// NETWORK 20
// label: (*IN1601 节能蓄能器气压*)
SaveEngine_PAtomsPre(
    INPUT := GVL_SaveEngine.AI_PAtomsPreMv,
    NEGFULL := PAR_HydOilPress_NegFull,
    POSFULL := PAR_HydOilPress_PosFull,
    RANGE := 400,
    Sensor_Error_LOW => CANO_SensorError_PAtomsPre,
    Sensor_Error_HIGH => CANO_SensorError_PAtomsPre); // PRESSURE
GVL_SaveEngine.AI_PAtomsPre := SaveEngine_PAtomsPre.OUTPUT;

// NETWORK 21
// IN 1602 主卷马达下降出口压力M1
SaveEngine_PM1Pre(
    INPUT := GVL_SaveEngine.AI_PM1PreMv,
    NEGFULL := PAR_HydOilPress_NegFull,
    POSFULL := PAR_HydOilPress_PosFull,
    RANGE := 400,
    Sensor_Error_LOW => CANO_SensorError_PM1,
    Sensor_Error_HIGH => CANO_SensorError_PM1); // PRESSURE
GVL_SaveEngine.AI_PM1Pre := SaveEngine_PM1Pre.OUTPUT;

// NETWORK 22
// IN 1603 主卷马达下降出口压力M2
SaveEngine_PM2Pre(
    INPUT := GVL_SaveEngine.AI_PM2PreMv,
    NEGFULL := PAR_HydOilPress_NegFull,
    POSFULL := PAR_HydOilPress_PosFull,
    RANGE := 400,
    Sensor_Error_LOW => CANO_SensorError_PM2,
    Sensor_Error_HIGH => CANO_SensorError_PM2); // PRESSURE
GVL_SaveEngine.AI_PM2Pre := SaveEngine_PM2Pre.OUTPUT;

// NETWORK 23 (disabled)
// Flow_Q1(Input := PI_Q1Freq, NEGFULL := 0, POSFULL := 2729, RANGE := 596); // Flow
// PI_Q1 := Flow_Q1.Output;

// NETWORK 24 (disabled)
// Flow_Q2(Input := PI_Q2Freq, NEGFULL := 0, POSFULL := 2729, RANGE := 596); // Flow
// PI_Q2 := Flow_Q2.Output;

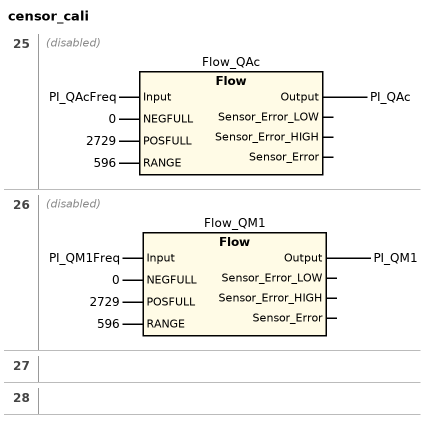
// NETWORK 25 (disabled)
// Flow_QAc(Input := PI_QAcFreq, NEGFULL := 0, POSFULL := 2729, RANGE := 596); // Flow
// PI_QAc := Flow_QAc.Output;

// NETWORK 26 (disabled)
// Flow_QM1(Input := PI_QM1Freq, NEGFULL := 0, POSFULL := 2729, RANGE := 596); // Flow
// PI_QM1 := Flow_QM1.Output;

// NETWORK 27

// NETWORK 28

END_FUNCTION_BLOCK

// StandardPLC/Application/CAIJI/ANGLE_CAIJI_X
FUNCTION_BLOCK ANGLE_CAIJI_X
VAR_INPUT
	input: UINT;
	negfull: UINT;
	zero: UINT;
	posfull: UINT;
END_VAR
VAR_OUTPUT
	output: INT;
	toollow: BOOL;
	toohigh: BOOL;
	Sensor_Error:BOOL;
END_VAR
VAR
	output1:DINT;
	output2: DINT;
END_VAR

IF(input<=0)  OR (input>65535)  THEN
	Sensor_Error:=TRUE;
ELSE
	Sensor_Error:=FALSE;
END_IF

IF input>posfull THEN
	output:=32767;
	toohigh:=TRUE;	toollow:=FALSE;
ELSIF input<negfull THEN
	output:=-32767;
	toohigh:=FALSE;	toollow:=TRUE;
ELSIF (input<=(zero+18) AND input>=(zero-18)) THEN
	output:=0;
	toohigh:=FALSE;	toollow:=FALSE;
ELSIF (input<(zero-18) AND input>=negfull) THEN
      output1:=UINT_TO_DINT(input)-UINT_TO_DINT(zero);
	IF output1<(-32767) THEN
		output:=-32767;
	ELSE
		output:=DINT_TO_INT(output1);
	END_IF
    IF (UINT_TO_REAL( input)-UINT_TO_REAL(zero))<-1460.0 THEN     (*x<4度*)
		toohigh:=FALSE;	toollow:=TRUE;
	ELSE
		toohigh:=FALSE;	toollow:=FALSE;
	END_IF
ELSIF (input>(zero+18) AND input<=posfull) THEN
	output2:=UINT_TO_DINT(input)-UINT_TO_DINT(zero);
	IF (output2>32767) THEN
		output:=32767;
	ELSE
		output:=DINT_TO_INT(output2);
	END_IF
     IF (UINT_TO_REAL( input)-UINT_TO_REAL(zero))>1460.0 THEN    (*1460=4度*)
		toohigh:=TRUE;	toollow:=FALSE;
	ELSE
		toohigh:=FALSE;	toollow:=FALSE;
	END_IF
ELSE
	output:=0;	toohigh:=FALSE;	toollow:=FALSE;
END_IF

END_FUNCTION_BLOCK

// StandardPLC/Application/CAIJI/ANGLE_CAIJI_Y
FUNCTION_BLOCK ANGLE_CAIJI_Y
VAR_INPUT
	input: UINT;
	negfull: UINT;
	zero: UINT;
	posfull: UINT;
END_VAR
VAR_OUTPUT
	output: INT;
	toohigh: BOOL;
	Sensor_Error:BOOL;
END_VAR
VAR
	output3: DINT;
	output4: DINT;
END_VAR

IF(input<=0)  OR (input>65535)  THEN
	Sensor_Error:=TRUE;
ELSE
	Sensor_Error:=FALSE;
END_IF

IF (UINT_TO_REAL( input)- UINT_TO_REAL(zero))>1460.0 THEN   (*y>4度*)
		toohigh:=TRUE;
ELSE
		toohigh:=FALSE;
END_IF

IF input>posfull THEN
	output:=32767;
ELSIF input<negfull THEN
	output:=-32767;
ELSIF (input<=(zero+18) AND input>=(zero-18)) THEN
	output:=0;
ELSIF (input<(zero-18) AND input>=negfull) THEN
	output3:=input-zero;
	IF output3<-32767 THEN
		output:=-32767;
	ELSE
		output:=DINT_TO_INT(output3);
	END_IF
ELSIF (input>(zero+18) AND input<=posfull) THEN
	output4:=input-zero;
	IF output4>32767 THEN
		output:=32767;
	ELSE
		output:=DINT_TO_INT(output4);
	END_IF
ELSE
	output:=0;
END_IF

END_FUNCTION_BLOCK

// StandardPLC/Application/CAIJI/HYD_OIL_TEM
FUNCTION_BLOCK HYD_OIL_TEM
VAR_INPUT
	Valt_Scale: UINT;
	Valt: UINT;
	In_Alarm_High:REAL;
END_VAR
VAR_OUTPUT
	Tem: REAL;
	Alarm_High:BOOL;
	Sensor_Error_TOOLOW:BOOL;
	Sensor_Error_TOOHIGH:BOOL;
END_VAR
VAR
	Ris: REAL;
END_VAR

Ris:=1000*UINT_TO_REAL(Valt)/UINT_TO_REAL(Valt_Scale);
IF Ris<168  THEN
	Tem:=85;
ELSIF Ris>=168 AND Ris<194 THEN
	Tem:=85+((Ris-168.0)*(80-85))/(194.0-168.0);
ELSIF Ris>=194 AND Ris<260 THEN
	Tem:=80+((Ris-194.0)*(70-80))/(260.0-194.0);
ELSIF Ris>=260 AND Ris<338 THEN
	Tem:=70+((Ris-260.0)*(60-70))/(338.0-260.0);
ELSIF Ris>=338 AND Ris<446 THEN
	Tem:=60+((Ris-338.0)*(50-60))/(446.0-338.0);
ELSIF Ris>=446 AND Ris<592 THEN
	Tem:=50+((Ris-446.0)*(40-50))/(592.0-446.0);
ELSIF Ris>=592 AND Ris<770 THEN
	Tem:=40+((Ris-592.0)*(30-40))/(770.0-592.0);
ELSIF Ris>=770 AND Ris<978 THEN
	Tem:=30+((Ris-770.0)*(20-30))/(978.0-770.0);
ELSE
	Tem:=20;
END_IF

IF Tem>In_Alarm_High THEN
	Alarm_High:=TRUE;
ELSE
	Alarm_High:=FALSE;
END_IF

IF Valt<=2   THEN
	Sensor_Error_TOOLOW:=TRUE;
ELSE
	Sensor_Error_TOOLOW:=FALSE;
END_IF
(*
IF Valt>=65000   THEN
	Sensor_Error_TOOHIGH:=TRUE;
ELSE
	Sensor_Error_TOOHIGH:=FALSE;
END_IF*)

END_FUNCTION_BLOCK

// StandardPLC/Application/CAIJI/FUEL_LEVEL
FUNCTION_BLOCK FUEL_LEVEL
VAR_INPUT
	INPUT: UINT;
	NEGFULL:UINT;
	POSFULL:UINT;
	In_Alarm_Low:UINT;
END_VAR
VAR_OUTPUT
	OUTPUT: UINT;
	Alarm_Low: BOOL;
	Sensor_Error_TOOLOW: BOOL;
	Sensor_Error_TOOHIGH: BOOL;
END_VAR
VAR
END_VAR

IF INPUT<=NEGFULL THEN
	INPUT:=NEGFULL;
ELSIF	INPUT>=POSFULL THEN
	INPUT:=POSFULL;
END_IF
OUTPUT:=REAL_TO_UINT((UINT_TO_REAL(INPUT-NEGFULL)/UINT_TO_REAL(POSFULL-NEGFULL))*100);
IF OUTPUT<In_Alarm_Low THEN
	Alarm_Low:=TRUE;
ELSE
	Alarm_Low:=FALSE;
END_IF

IF INPUT<=2 THEN
	Sensor_Error_TOOLOW:=TRUE;
ELSE
	Sensor_Error_TOOLOW:=FALSE;
END_IF
IF INPUT>=65000 THEN
	Sensor_Error_TOOHIGH:=TRUE;
ELSE
	Sensor_Error_TOOHIGH:=FALSE;
END_IF

END_FUNCTION_BLOCK

// StandardPLC/Application/CAIJI/PRESSURE
FUNCTION_BLOCK PRESSURE
VAR_INPUT
	INPUT: UINT;
	NEGFULL:UINT;
	POSFULL:UINT;
	RANGE:UINT;
END_VAR
VAR_OUTPUT
	OUTPUT: UINT;
	Sensor_Error_LOW: BOOL;
	Sensor_Error_HIGH:BOOL;
	Sensor_Error: BOOL;
END_VAR

IF INPUT<=NEGFULL THEN
	INPUT:=NEGFULL;
ELSIF	INPUT>=POSFULL THEN
	INPUT:=POSFULL;
ELSE
	OUTPUT:=REAL_TO_UINT((UINT_TO_REAL(INPUT-NEGFULL)/UINT_TO_REAL(POSFULL-NEGFULL))*UINT_TO_REAL(RANGE));
END_IF

IF  INPUT<=3800  THEN
	Sensor_Error_LOW:=TRUE;
ELSE
	Sensor_Error_LOW:=FALSE;
END_IF

IF  INPUT>=20000  THEN
	Sensor_Error_HIGH:=TRUE;
ELSE
	Sensor_Error_HIGH:=FALSE;
END_IF

IF Sensor_Error_LOW OR Sensor_Error_HIGH THEN
	Sensor_Error := TRUE;
ELSE
	Sensor_Error := FALSE;
END_IF

END_FUNCTION_BLOCK

// StandardPLC/Application/CAIJI/Tension
FUNCTION_BLOCK Tension
VAR_INPUT
	INPUT: UINT;
	NEGFULL:UINT;
	POSFULL:UINT;
	Coefficient:REAL;
	RANGE:UINT;
END_VAR
VAR_OUTPUT
	OUTPUT: UINT;
	Sensor_Error_LOW: BOOL;
	Sensor_Error_HIGH:BOOL;
	Sensor_Error: BOOL;
END_VAR
VAR
END_VAR

IF INPUT<=NEGFULL THEN
	INPUT:=NEGFULL;
ELSIF	INPUT>=POSFULL THEN
	INPUT:=POSFULL;
ELSE
	OUTPUT:=REAL_TO_UINT(10*0.6*(UINT_TO_REAL(INPUT-NEGFULL)/UINT_TO_REAL(POSFULL-NEGFULL))*UINT_TO_REAL(RANGE));
END_IF

IF  INPUT<=3800  THEN
	Sensor_Error_LOW:=TRUE;
ELSE
	Sensor_Error_LOW:=FALSE;
END_IF

IF  INPUT>=20000  THEN
	Sensor_Error_HIGH:=TRUE;
ELSE
	Sensor_Error_HIGH:=FALSE;
END_IF

IF Sensor_Error_LOW OR Sensor_Error_HIGH THEN
	Sensor_Error := TRUE;
ELSE
	Sensor_Error := FALSE;
END_IF

END_FUNCTION_BLOCK

// StandardPLC/Application/MOVE/worktime
PROGRAM worktime
VAR
	init_TIME:BOOL:=TRUE;
	counter1: UINT;
	minute: UDINT;
	work_time: UDINT;
	x:BLINK;
    A:ARRAY[1..40] OF BYTE;
	b:BOOL;
	SHIJIAN:TON;
	T_TP: TP;
	XIANWEI: BOOL;
	TEMP1:DWORD;
	RTIG:F_TRIG;
	RTRIG1:R_TRIG;
	COUNT2: INT;
END_VAR

IF init_TIME THEN
	Mid_worktime:=PAR_WorkTime;
	init_TIME:=FALSE;
END_IF

IF CANO_SPEED>200  THEN
	SHIJIAN(IN:=TRUE,PT:=T#999h9m);
	TEMP1:=TIME_TO_DWORD(SHIJIAN.ET);
	minute:=TEMP1/60000;
	PAR_WorkTime:=Mid_worktime+minute;
END_IF

CANO_engine_hour_h:=TO_DINT(PAR_WorkTime/60);
CANO_engine_hour_m:=UDINT_TO_BYTE(PAR_WorkTime MOD 60);

IF CANI_Button_RecordClear THEN
	PAR_WorkTime:=0;
	Mid_worktime:=0;
END_IF

IF(NOT CANI_WorkModeSwitch)AND(CANI_JOY_SB2)AND(CANI_JOY_SB1)THEN
	PAR_DISTANCE_CANCEL:=TRUE;
ELSE
	PAR_DISTANCE_CANCEL:=FALSE;
END_IF

(*BUZZER*)
IF(NOT	CANI_Button_BuzzSwitch)THEN
	IF(CANO_TooLow_BatteryVol AND CANO_SPEED>500 )OR(CANO_TooLow_FUEL_LEVEL)OR(CANO_TooHigh_HydOilTem)OR(CANO_TooHigh_WaterTem)OR(CANO_TooLow_OilPress AND CANO_SPEED>200)
		OR(DIL_SQ4)OR(DIH_SP4)THEN
		DOH_B1:=TRUE;
	ELSE
		DOH_B1:=FALSE;
	END_IF
ELSIF(CANI_Button_BuzzSwitch)THEN
	DOH_B1:=FALSE;
END_IF
(*限位模式*)
IF(NOT DIH_SQ5)THEN
	CANO_LimiteModle:=2;
ELSIF(NOT DIH_SQ6)THEN
	CANO_LimiteModle:=1;
ELSE
	CANO_LimiteModle:=0;
END_IF
IF(PAR_ControlValue=9999)THEN
	CANO_Limite_Cancel:=TRUE;
ELSE
	CANO_Limite_Cancel:=FALSE;
END_IF

IF AI_SP1>4990 THEN
	AI_SP1:=4990;
END_IF

IF AI_JOYX>4880 THEN
	AI_JOYX:=4880;
END_IF

IF AI_JOYY>4880 THEN
	AI_JOYY:=4880;
END_IF
(*油温控制*)
(*温度超过60度时，风扇自动打开，温度低于50度时，风扇自动关闭*)
IF CANO_Hyd_Tem>60  THEN
	DOH_Y57:=FALSE;
ELSIF CANO_Hyd_Tem<50  THEN
	DOH_Y57:=TRUE;
END_IF

IF CANI_ColdFunSwitch THEN
	DOH_Y57:=FALSE;
END_IF
(*液压手柄电子锁定*)
RTRIG1(CLK:=CANI_JOY_SB7);
(*液压油温限值*)
(*液压油温限值*)
IF(AI_SP3<=5000)THEN
	AI_SP3_1:=AI_SP3;
ELSE
	AI_SP3_1:=5000;
END_IF

IF(AI_SP1<=5000)THEN
	AI_SP1_1:=AI_SP1;
ELSE
	AI_SP1_1:=5000;
END_IF

END_PROGRAM

// StandardPLC/Application/CAIJI/ZONGXIANJISUAN
FUNCTION_BLOCK ZONGXIANJISUAN
VAR_INPUT
END_VAR
VAR_OUTPUT
	X:UINT;
	Y:UINT;
	ERROR:BOOL;
END_VAR
VAR
	CAN2RECEIVE_1FF:ifmRCAN.CAN_Rx;
	receive_data1FF:ARRAY [0..7] OF USINT;
	A:UINT;
	B:UINT;
END_VAR

CAN2RECEIVE_1FF(xEnable:=TRUE , eChannel:= 1, xExtended:= FALSE, aData=> receive_data1FF, udiID:= 16#1FF);
A:=USINT_TO_UINT(receive_data1FF[0])+256*USINT_TO_UINT(receive_data1FF[1]);
B:=USINT_TO_UINT(receive_data1FF[2])+256*USINT_TO_UINT(receive_data1FF[3]);

IF(A>=0)AND(A<=1800)THEN
	X:=REAL_TO_UINT(UINT_TO_REAL(A)/3600.0*65535+32767);
END_IF
IF(A>=63735)AND(A<=65535)THEN
	X:=REAL_TO_UINT(32767-(65535-UINT_TO_REAL(A))/3600.0*65535);
END_IF
IF(B>=0)AND(B<=1800)THEN
	Y:=REAL_TO_UINT(UINT_TO_REAL(B)/3600.0*65535+32767);
END_IF
IF(B>=63735)AND(B<=65535)THEN
	Y:=REAL_TO_UINT(32767-(65535-UINT_TO_REAL(B))/3600.0*65535);
END_IF
IF receive_data1FF[0]=16#FF AND  receive_data1FF[1]=16#FF AND receive_data1FF[2]=16#FF AND receive_data1FF[3]=16#FF THEN
	ERROR:=TRUE;
ELSE
	ERROR:=FALSE;
END_IF

(*(*采用电流型输入的倾角传感器4-20mA*)
IF(AI_AngleX>12000 AND AI_AngleX<=20000) THEN
	A:=REAL_TO_UINT((UINT_TO_REAL(AI_AngleX)-12000)*1800/8000);
ELSIF (AI_AngleX>=4000 AND AI_AngleX<=12000) THEN
	A:=REAL_TO_UINT(65535-(12000-UINT_TO_REAL(AI_AngleX))*1800/8000);
END_IF

IF(AI_AngleY>12000 AND AI_AngleY<=20000) THEN
	B:=REAL_TO_UINT((UINT_TO_REAL(AI_AngleY)-12000)*1800/8000);
ELSIF (AI_AngleY>=4000 AND AI_AngleY<=12000) THEN
	B:=REAL_TO_UINT(65535-(12000-UINT_TO_REAL(AI_AngleY))*1800/8000);
END_IF

IF(A>=0)AND(A<=1800)THEN
	X:=REAL_TO_UINT(UINT_TO_REAL(A)/3600.0*65535+32767);//32768-65535 表示0-90°
END_IF
IF(A>=63735)AND(A<=65535)THEN
	X:=32767-REAL_TO_UINT(UINT_TO_REAL(65535-A)/3600.0*65535);//0-32767 表示-90°-0°
END_IF
IF(B>=0)AND(B<=1800)THEN
	Y:=REAL_TO_UINT(UINT_TO_REAL(B)/3600.0*65535+32767);//32768-65535 表示0-90°
END_IF
IF(B>=63735)AND(B<=65535)THEN
	Y:=32767-REAL_TO_UINT(UINT_TO_REAL(65535-B)/3600.0*65535);//0-32767 表示-90°-0°
END_IF
(*IF receive_data1FF[0]=16#FF AND  receive_data1FF[1]=16#FF AND receive_data1FF[2]=16#FF AND receive_data1FF[3]=16#FF THEN
	ERROR:=TRUE;
ELSE
	ERROR:=FALSE;
END_IF*)

IF AI_AngleX<4000 OR AI_AngleX>20000 OR AI_AngleY<4000 OR AI_AngleY>20000 THEN
	ERROR:=TRUE;
ELSE
	ERROR:=FALSE;
END_IF*)

END_FUNCTION_BLOCK

// StandardPLC/Application/CAIJI/CAN_XY
FUNCTION_BLOCK CAN_XY
VAR_INPUT
	sensor_x:UINT;
	sensor_y:UINT;
END_VAR
VAR_OUTPUT
	CAN_X:UINT;
	CAN_Y:UINT;
	CAN_XY_Q:BOOL;
END_VAR
VAR
END_VAR

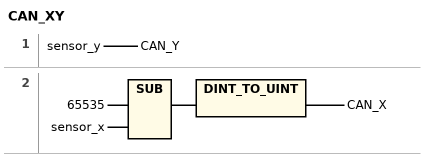
// NETWORK 1
CAN_Y := sensor_y;

// NETWORK 2
CAN_X := DINT_TO_UINT(65535 - sensor_x);

END_FUNCTION_BLOCK

// StandardPLC/Application/CAIJI/CAIJI_DEPTH
PROGRAM CAIJI_DEPTH
VAR
	depth_a: DEPTH;
	DEPTH1: UINT;
	TIME_1000ms:TON;
	TM:DWORD;
	TM_OLD:TIME;
(*速度计算*)
	depth_neij1: UINT;
	i:UINT;
	H:UINT;
	R_trig1:R_TRIG;
	R_trig2:R_TRIG;
	Mid_Depth_Value:DINT;
	MM_Depth_Value:DINT;
	Mid_Value: DINT;
	Total_Value: REAL;
	MainWinch_Speed_M:REAL;
END_VAR


	depth_a(DEPTH_A:=DIH_SQ1,DEPTH_B:=DIH_SQ2,reset:=CANI_Button_DepthClear);
	DEPTH:=REAL_TO_INT(DINT_TO_REAL(IncEncoder_temp_diValue)/96.0*(3.14*UINT_TO_REAL(PAR_Circle2))/10.0);
	(*DEPTH:=REAL_TO_INT(DINT_TO_REAL(PI_Depth_COUNTER)/96.0*(3.14*UINT_TO_REAL(PAR_Circle2))/10.0);*)
	IF(DEPTH<-1000) THEN
		DEPTH := -1000;
	END_IF
	DEPTH1:=INT_TO_UINT(DEPTH+1000);
	CANO_DEPTH:=DEPTH1;
	
	IF(PAR_DEPTH_VALUE<DEPTH1)THEN   //上次孔深
		PAR_DEPTH_VALUE:=DEPTH1;
	END_IF
	
	IF(CANO_DEPTH<PAR_DEPTH_VALUE)THEN
		PAR_DEPTH_VALUE2:=PAR_DEPTH_VALUE;
	END_IF
	
(***************卷扬速度计算***************)
	TIME_1000ms(IN:=(i>0),PT:=T#1M);
	i:=i+1;
	R_trig1(CLK:=(i=1));
	IF ( i MOD 10)=0 AND  i>1 THEN
		Mid_Value:=(DEPTH-MM_Depth_Value);
		Total_Value:=Total_Value+DINT_TO_REAL(Mid_Value);//每10个循环更新一次累计位移差值
	END_IF

	IF i=100 THEN//100个循环计算一次速度,一个循环10ms,1s更新一次速度  //1s-200ms  20-100 2024 0125
		MainWinch_Speed:=REAL_TO_INT(Total_Value*(60.0/(( TIME_TO_REAL(TIME_1000ms.ET))/1000.0)));//每分钟的位移量，m/min
	  		  i:=0;
			Total_Value:=0;
			Mid_Value:=0;
	END_IF

	IF R_Trig1.Q  OR (( i MOD 10)=0 AND  i>1)  THEN
		MM_Depth_Value:=DEPTH;
	END_IF

	CANO_MainWinch_Speed:=INT_TO_UINT(MainWinch_Speed / 10 + 1000);
	MainWinch_Speed_M:= UINT_TO_INT(CANO_MainWinch_Speed-1000)/10;
(***************累计深度计算***************)
	//累计钻孔深度的计算
	IF(VarDepthLastMax<=CANO_DEPTH) THEN
		VarDepthLastMax := CANO_DEPTH;//接收孔深最大值
	END_IF
	
	VarMaiWinDepth_subtract := UINT_TO_DINT(CANO_DEPTH) - UINT_TO_DINT(VarDepthLastMax);
	
	IF(VarMaiWinDepth_subtract < 0)THEN
		VarMaiWinDepth_Up_biaozhi := TRUE;
	ELSE
		VarMaiWinDepth_Up_biaozhi := FALSE;
	END_IF

	IF((VarMaiWinDepth_Up_biaozhi) AND (VarMaiWinDepthLast<VarDepthLastMax))THEN
		VarMaiWinDepthOnce := VarDepthLastMax - VarMaiWinDepthLast;
		VarMaiWinDepthLast := VarDepthLastMax;
	END_IF

	IF(VarMaiWinDepthOnce>0)THEN
		DEPTH_accumu:=DEPTH_accumu + VarMaiWinDepthOnce;
		VarMaiWinDepthOnce :=0;
	END_IF

	CANO_ACCMUDEPTH:=DEPTH_accumu;

END_PROGRAM

// StandardPLC/Application/CAIJI/DEPTH
FUNCTION_BLOCK DEPTH
VAR_INPUT
	DEPTH_A: BOOL;
	DEPTH_B: BOOL;
	reset: BOOL;
END_VAR
VAR_OUTPUT
	DEPTH_PI: INT;
END_VAR
VAR
	Q0: BOOL;
	M0: BOOL := TRUE;
	Q1: BOOL;
	Q2: BOOL;
	M1: BOOL := TRUE;
	M2: BOOL := TRUE;
	Q3: BOOL;
	M3: BOOL := TRUE;

	Q: BOOL;
	f1: BOOL;
	f2: BOOL;
	f0: BOOL;
	f3: BOOL;
	cf0: BOOL;
	cf1: BOOL;
	cf2: BOOL;
	cf3: BOOL;
	CW_R:BOOL;
	CCW_R:BOOL;
	CWrt:R_TRIG;
	CcWrt:R_TRIG;

	PI_SQ1_1: DINT;
	PI_SQ1_2: DINT;
	PI_SQ2_1: DINT;
	PI_SQ2_2: DINT;
	PI_SQ1_REAL: DINT;
	PI_SQ2_REAL:DINT;
	
	PI_SQ1_3:DINT;
	PI_SQ1_4:DINT;
	PI_SQ2_3:DINT;
	PI_SQ2_4:DINT;
	
END_VAR

Q0:=DEPTH_A  AND NOT M0;
M0:=DEPTH_A;
Q1:=DEPTH_B AND NOT M1;
M1:=DEPTH_B;
Q2:=NOT DEPTH_A  AND NOT M2;
M2:=NOT DEPTH_A;
Q3:=NOT DEPTH_B  AND NOT M3;
M3:=NOT DEPTH_B;
Q:=Q0 OR Q1 OR Q2 OR Q3;

f0:=Q0 AND NOT DEPTH_B;
f1:=Q1 AND DEPTH_A;
f2:=Q2 AND DEPTH_B;
f3:=Q3 AND NOT DEPTH_A;
cf0:=Q1 AND (NOT DEPTH_A);
cf1:=Q0 AND DEPTH_B;
cf2:=Q3 AND DEPTH_A;
cf3:=Q2 AND (NOT DEPTH_B);
(*IF f0 OR f1 OR f2 OR f3 THEN
	CW:=TRUE;
	CCW:=FALSE;
ELSIF cf0 OR cf1 OR cf2 OR cf3 THEN
	CCW:=TRUE;
	CW:=FALSE;
END_IF
IF CW AND Q THEN
	DEPTH_PI:=DEPTH_PI+1;
ELSIF CCW AND Q THEN
	DEPTH_PI:=DEPTH_PI-1;
END_IF*)

IF (* PWM_JOYY_L_DOWN>10 OR *)(PWM_Y7>610  OR PWM_Y9>610)   THEN   //主卷上提时
	CW:=FALSE;
	CCW:=TRUE;
ELSIF (*PWM_JOYY_L_UP>10 OR*) (PWM_Y8>610 OR PWM_Y10>610 )OR DOH_Y56 THEN   //主卷下放时
	CW:=TRUE;
	CCW:=FALSE;
ELSE
	CW:=FALSE;
	CCW:=FALSE;
END_IF


CWrt(CLK:=CW,Q=>CW_R);
CcWrt(CLK:=CCW,Q=>CCW_R);

IF CW_R THEN   //正转上升沿时
 PI_SQ1_1:=TO_DINT(PI_SQ1);
 PI_SQ1_2:=PI_SQ1_REAL;
 PI_SQ2_1:=TO_DINT(PI_SQ2);
 PI_SQ2_2:=PI_SQ2_REAL;
END_IF
IF CW THEN  //
 PI_SQ1_REAL:=PI_SQ1_2+(TO_DINT(PI_SQ1)-PI_SQ1_1);
 PI_SQ2_REAL:=PI_SQ2_2+(TO_DINT(PI_SQ2)-PI_SQ2_1);
END_IF
IF CCW_R THEN   //反转上升沿时
 PI_SQ1_3:=TO_DINT(PI_SQ1);
 PI_SQ1_4:=PI_SQ1_REAL;
 PI_SQ2_3:=TO_DINT(PI_SQ2);
 PI_SQ2_4:=PI_SQ2_REAL;
END_IF
IF CCW THEN
 PI_SQ1_REAL:=PI_SQ1_4-(TO_DINT(PI_SQ1)-PI_SQ1_3);
 PI_SQ2_REAL:=PI_SQ2_4-(TO_DINT(PI_SQ2)-PI_SQ2_3);
END_IF
DEPTH_PI:=TO_INT(PI_SQ1_REAL+PI_SQ2_REAL);



IF reset THEN
	Tmp_Depth:=0;
	PAR_DEPTH_VALUE:=0;
	VarMaiWinDepthLast:=1000;
	VarDepthLastMax:=1000;
	VarMaiWinDepthOnce:=0;
	PI_SQ1_1:=0;
	PI_SQ1_2:=0;
	PI_SQ2_1:=0;
	PI_SQ2_2:=0;
	PI_SQ1_3:=0;
	PI_SQ1_4:=0;
	PI_SQ2_3:=0;
	PI_SQ2_4:=0;
	PI_SQ1_REAL:=0;
	PI_SQ2_REAL:=0;
	DEPTH_PI:=0;
END_IF
IF CANI_Button_RecordClear  THEN
	DEPTH_accumu:=0;
	PAR_DEPTH_accumu:=0;
	PAR_DEPTH_VALUE:=0;
	DEPTH_PI:=0;
	Tmp_Depth:=0;
	VarMaiWinDepthLast:=1000;
	VarDepthLastMax:=1000;
	VarMaiWinDepthTotal:= 0;
END_IF

END_FUNCTION_BLOCK

// StandardPLC/Application/MOVE/MODE_ROTATE
FUNCTION_BLOCK MODE_ROTATE
VAR_INPUT
END_VAR
VAR_OUTPUT
	MODE_ROTATE_AU: BOOL;
	MODE_ROTATE_MA: BOOL;
END_VAR
VAR
	num:UINT;
	RTRIGLnst:R_TRIG;

	A: BOOL;
	B: UINT;

	TIAOJIAN: BOOL;

END_VAR

IF (DI_LHandle_SB7)  THEN
	MODE_ROTATE_AU:=TRUE;
	MODE_ROTATE_MA:=FALSE;
ELSE
	MODE_ROTATE_MA:=TRUE;
	MODE_ROTATE_AU:=FALSE;
END_IF

CANO_RotationModle:=MODE_ROTATE_AU;

END_FUNCTION_BLOCK

// StandardPLC/Application/MOVE/ROTATE_AUTO
FUNCTION_BLOCK ROTATE_AUTO
VAR_INPUT
	CON_IROTATE:UINT;
	MODE_ROTATE_AU:BOOL;
	MODE_ROTATE_MA:BOOL;

END_VAR
VAR_OUTPUT
	CON_OROTATE:INT;
END_VAR
VAR
	TIAOJIAN: BOOL;
	step: INT;
	control:INT:=0;
	e1:INT;
	e2:INT;
	e3:INT;
	A1:BOOL;
	A2:R_TRIG;
	par_k:UINT:=10000;

END_VAR

IF(CANO_DEPTH<950)THEN
	TIAOJIAN:=TRUE;
ELSE
	TIAOJIAN:=FALSE;
END_IF
e3:=e2;
e2:=e1;
e1:=UINT_TO_INT(CON_IROTATE);

(*par_sudu1_min为正向最小控制量，par_sudu1_max为正向最大控制量，par_sudu1_zhong为中间控制量par_angle1为正向最小脉冲值，    *)
(*par_angle2 为下降控制量时的脉冲值  par_angle3为中间下降脉冲值*)
IF MODE_ROTATE_AU AND TIAOJIAN THEN
	IF(CON_IROTATE>=par_angle2 AND CON_IROTATE<=2048)THEN		  (*此过程为加速过程至最大值*)
		step:=REAL_TO_INT((INT_TO_REAL(UINT_TO_INT(par_sudu1_max))-INT_TO_REAL(UINT_TO_INT(par_sudu1_min)))/100);
		IF(control<UINT_TO_INT(par_sudu1_max))THEN
			control:=control+step;
		ELSIF (control>=UINT_TO_INT(par_sudu1_max))  THEN
			control:=UINT_TO_INT(par_sudu1_max);
		END_IF
	END_IF
	IF(CON_IROTATE>=par_angle3 AND CON_IROTATE<par_angle2 )THEN   (*此过程为从最大速度减速至中速*)
			step:=REAL_TO_INT((INT_TO_REAL(UINT_TO_INT(par_sudu1_max))-INT_TO_REAL(UINT_TO_INT(par_sudu1_min)))/100);
		IF(control>UINT_TO_INT(PAR_Sudu1_Middle)) THEN
			control:=control-step;
		ELSIF(control<=UINT_TO_INT(PAR_Sudu1_Middle)) THEN
			control:=UINT_TO_INT(PAR_Sudu1_Middle);
		END_IF
	END_IF
	IF(CON_IROTATE>=par_angle1 AND CON_IROTATE<par_angle3)THEN
			step:=REAL_TO_INT((INT_TO_REAL(UINT_TO_INT(par_sudu1_max))-INT_TO_REAL(UINT_TO_INT(par_sudu1_min)))/100);
		IF(control>UINT_TO_INT(par_sudu1_min)) THEN
			control:=control-step;
		ELSIF(control<=UINT_TO_INT(par_sudu1_min)) THEN
			control:=UINT_TO_INT(par_sudu1_min);
		END_IF
	END_IF
	IF(CON_IROTATE>=0 AND CON_IROTATE<par_angle1 )THEN
		IF(CON_IROTATE>3)THEN
			IF ABS(UINT_TO_INT(CON_IROTATE)) <=UINT_TO_INT(par_k)*ABS(e3-UINT_TO_INT(CON_IROTATE)) THEN
				control:=0;
				A1:=TRUE;
				A2(CLK:=A1);
				CANO_ZHIXING:=A2.Q;
			ELSE
				control:=UINT_TO_INT(par_sudu1_min);
				CANO_ZHIXING:=0;
			END_IF
		END_IF
		IF(CON_IROTATE<=3)THEN
			control:=0;
		END_IF
	END_IF
(*FUXIANG*)
(*par_sudu2_min为反向最小控制量，par_sudu2_max为反向最大控制量，par_angle5为下降控制量时的脉冲值，    par_angle4为反向最小脉冲值
par_sudu2_zhong为中间控制量  par_angle6为中间脉冲值*)
	IF(CON_IROTATE>2048 AND CON_IROTATE<=par_angle5)THEN
			step:=REAL_TO_INT((INT_TO_REAL(-UINT_TO_INT(par_sudu2_max))+INT_TO_REAL(UINT_TO_INT(par_sudu2_min)))/100);
		IF((control)>(-UINT_TO_INT(par_sudu2_max))) THEN
			control:=control+step;
		ELSIF (control)<=(-UINT_TO_INT(par_sudu2_max))  THEN
			control:=-UINT_TO_INT(par_sudu2_max);
		END_IF
	END_IF
	IF(CON_IROTATE>par_angle5 AND CON_IROTATE<=par_angle6 )THEN
			step:=REAL_TO_INT((INT_TO_REAL(-UINT_TO_INT(par_sudu2_max))+INT_TO_REAL(UINT_TO_INT(par_sudu2_min)))/100);
		IF (control)<(-UINT_TO_INT(PAR_Sudu2_Middle)) THEN
			control:=control-step;
		ELSIF(control)>=(-UINT_TO_INT(PAR_Sudu2_Middle)) THEN
			control:=-UINT_TO_INT(PAR_Sudu2_Middle);
		END_IF
	END_IF
	IF(CON_IROTATE>par_angle6 AND CON_IROTATE<=par_angle4 )THEN
			step:=REAL_TO_INT((INT_TO_REAL(-UINT_TO_INT(par_sudu2_max))+INT_TO_REAL(UINT_TO_INT(par_sudu2_min)))/100);
		IF(control)<(-UINT_TO_INT(par_sudu2_min))THEN
			control:=control-step;
		ELSIF(control)>=(-UINT_TO_INT(par_sudu2_min))THEN
			control:=-UINT_TO_INT(par_sudu2_min);
		END_IF
	END_IF
	IF(CON_IROTATE>par_angle4 AND CON_IROTATE<=4096 )THEN
		IF(CON_IROTATE<4093)THEN
			IF ABS(4096-UINT_TO_INT(CON_IROTATE))<=UINT_TO_INT(par_k)*ABS(e3-UINT_TO_INT(CON_IROTATE))THEN
				control:=0;
				A1:=TRUE;
				A2(CLK:=A1);
				CANO_ZHIXING:=A2.Q;
			ELSE
				control:=-UINT_TO_INT(par_sudu2_min);
				CANO_ZHIXING:=0;
			END_IF
		END_IF
		IF(CON_IROTATE>=4093)THEN
			control:=0;
		END_IF
	END_IF
ELSE
control:=0;
END_IF
CON_OROTATE:=control;

END_FUNCTION_BLOCK

// StandardPLC/Application/SaveEngine/Wt_Cal
PROGRAM Wt_Cal
VAR
	MainWinchTension_M:REAL;
	
	MainWinchTension_Sum1:UINT:=0;
	MainWinchTension1:ARRAY[0..200] OF UINT;
	m1: UINT:=200;	
	MainWinchTension_i1:UINT;
	MainWinchTension_Ave1:REAL;
END_VAR

MainWinchTension_Sum1:=0;
MainWinchTension1[m1]:=CANO_MainWinchTension;
FOR MainWinchTension_i1:=0 TO (m1-1) BY 1 DO
	MainWinchTension1[MainWinchTension_i1]:=MainWinchTension1[MainWinchTension_i1+1];
	MainWinchTension_Sum1:=MainWinchTension_Sum1+MainWinchTension1[MainWinchTension_i1];
END_FOR
MainWinchTension_Ave1:= (MainWinchTension_Sum1)/(m1);


//IF DEPTH <= 0 AND PWM_JOYY_L_DOWN<300 AND PWM_JOYY_L_UP<300 THEN
IF DEPTH <= 0 AND PWM_JOYY_L_DOWN<500 AND PWM_JOYY_L_UP<500 THEN
	MainWinchTension_M:=MainWinchTension_Ave1;
	IF  MainWinchTension_M > Max_MainWinchTension THEN
		Max_MainWinchTension:=MainWinchTension_M;
	END_IF
END_IF

END_PROGRAM

// StandardPLC/Application/MOVE/inti_fasle
PROGRAM inti_fasle
VAR
END_VAR

init_1:=FALSE;
init_2:=FALSE;

END_PROGRAM

// StandardPLC/Application/MOVE/PID_JYF
FUNCTION_BLOCK PID_JYF
VAR_INPUT
	MeasPoint: INT;
	SetPoint: INT;
	P:UINT;
	I: REAL;
	D: USINT;
	RC: USINT;
	ENABLE: BOOL;
	RAMP: UINT;
END_VAR
VAR_OUTPUT
	Control: DINT;
END_VAR
VAR
	E: INT;
	E1: INT;
	E2: INT;
	COUNTER: UINT;
END_VAR

IF (RAMP<=COUNTER) THEN
	IF(ENABLE)THEN
		E:=E+(SetPoint-MeasPoint-E)/RC;
		Control:=REAL_TO_DINT(DINT_TO_REAL(Control)+(E-E1)*UINT_TO_INT(P)/10+E*I/5+(E-2*E1+E2)*D/10);
		E2:=E1;
		E1:=E;
	IF (Control<-32767) THEN
		Control:=-32767;
	END_IF

	IF (Control>32767) THEN
		Control:=32767;
	END_IF
	ELSE
		E:=0;
		E1:=0;
		E2:=0;
		Control:=0;
	END_IF
	COUNTER:=0;
ELSE
	COUNTER:=COUNTER+1;
END_IF

END_FUNCTION_BLOCK

// Project Information/GetVersion
// This function has been automatically generated from the project information.
{attribute 'signature_flag' := '1073741824'}
{attribute 'register_in_runtime'}
FUNCTION GetVersion : VERSION
VAR_INPUT
	
END_VAR

GetVersion.uiMajor := 3;
GetVersion.uiMinor := 1;
GetVersion.uiServicePack := 4;
GetVersion.uiPatch := 1;

END_FUNCTION

// Project Information/GetCompany
// This function has been automatically generated from the project information.
{attribute 'signature_flag' := '1073741824'}
{attribute 'register_in_runtime'}
FUNCTION GetCompany : WSTRING
VAR_INPUT
	
END_VAR

GetCompany := "ifm electronic";

END_FUNCTION

// Project Information/GetTitle
// This function has been automatically generated from the project information.
{attribute 'signature_flag' := '1073741824'}
{attribute 'register_in_runtime'}
FUNCTION GetTitle : WSTRING
VAR_INPUT
	
END_VAR

GetTitle := "ifmCR721S_TemplateProject";

END_FUNCTION

// Project Information/GetTextProperty2
// This function has been automatically generated from the project information.
{attribute 'signature_flag' := '1073741824'}
{attribute 'register_in_runtime'}
FUNCTION GetTextProperty2 : POINTER TO WSTRING
VAR_INPUT
	stKey: WSTRING;
END_VAR

IF stKey = "Company" THEN
	GetTextProperty2 := ADR("ifm electronic");
ELSIF stKey = "Description" THEN
	GetTextProperty2 := ADR("CR721S 2.25MByte Standard and Safety");
ELSIF stKey = "Project" THEN
	GetTextProperty2 := ADR("SWDM240HES_S00107_20240126_Y33");
ELSIF stKey = "Title" THEN
	GetTextProperty2 := ADR("ifmCR721S_TemplateProject");
ELSE
	GetTextProperty2 := ADR("");
END_IF

END_FUNCTION

// StandardPLC/Application/CAN/GPS_ALL
PROGRAM GPS_ALL
VAR
		send_data300:ARRAY [0..7] OF USINT;	
		send_data300_1:ARRAY [0..7] OF USINT;
		send_data18FF0001: ARRAY [0..7] OF USINT;
		CAN2_SEND_300:ifmRCAN.CAN_Tx;
		CAN2_SEND_18FF00001:ifmRCAN.CAN_Tx;
		CAN2_RECE_GPS200:ifmRCAN.CAN_Rx;
		receive_data200:ARRAY [0..7] OF USINT;
		archives:UINT;
		X_Offset_zhongjian: REAL;
		Y_Offset_zhongjian: REAL;
		Y_Offset: UINT;
		X_Offset: UINT;
		TIME_5S:TON;
		TIME_1S:TON;
		TIME_1S_1:TON;
		TIME_600S:TON;
		TIME_600S_2:TON;
		TIME_60s:TON;
		TIME_60s_2:TON;
		TIME_2s:TON;
		temp:USINT;
		tU8_L:USINT;
		tU8_H :USINT;
		tU16:UINT;
		GPS_CAN_ERROR_1: BOOL;
		GPSYONGJIU:TMP.Passward;
		
		
		
		

END_VAR

(*控制器向GPS发送数据*)
archives := archives + 1;
IF archives>22  THEN
	archives := 0;
END_IF
TIME_5S(In:= NOT TIME_5S.Q,Pt:=T#5S);(*每5s钟00/01跳变*)
IF TIME_5S.Q THEN
	temp:=temp+1;
END_IF
CASE archives OF
	0:(*组合向GPS发送的新版协议数据,序号0x00*)
		send_data300_1[0]:=16#00;
		send_data300_1[1]:=temp MOD 2;(*每5s钟00/01跳变*)
		send_data300_1[2]:=00;
		send_data300_1[3]:=06;(*通讯协议版本号*)
		send_data300_1[4]:=0;
		send_data300_1[5]:=0;
		send_data300_1[6]:=0;
		send_data300_1[7]:=0;
	1:(*组合向GPS发送的新版协议数据,序号0x01*)
		send_data300_1[0]:=16#01;
		send_data300_1[1]:=PACK(B0:=VarGpsGlobalEnable,B1:=NOT VarGpsGlobalEnable,B2:=VarGpsTempUnlockDoing,B3:= VarGpsPasswordTempUnlockEnable,B4:=0,B5:=0,B6:=0,B7:=0);
		send_data300_1[2]:=0;
		send_data300_1[3]:=0;
		send_data300_1[4]:=UDINT_TO_USINT((VarGpsPasswordTemporaryCode MOD 65536) MOD 256);
		send_data300_1[5]:=UDINT_TO_USINT((VarGpsPasswordTemporaryCode MOD 65536) /256);
		send_data300_1[6]:=UDINT_TO_USINT((VarGpsPasswordTemporaryCode / 65536) MOD 256);
		send_data300_1[7]:=UDINT_TO_USINT((VarGpsPasswordTemporaryCode / 65536)/256);
	2:(*组合向GPS发送的新版协议数据,序号0x02*)
		send_data300_1[0]:=16#02;
		send_data300_1[1]:=PACK(B0:=VarCanGpsKongZhiQiLockCommand AND VarGpsSystemLockedState,
								B1:=0,
								B2:=VarCanGpsYanShiLockCommand AND VarGpsSystemLockedState,
								B3:= VarCanGpsTianXianLockCommand AND VarGpsSystemLockedState,
								B4:=VarCanGpsKaiGaiLockCommand AND VarGpsSystemLockedState ,
								B5:=VarCanGpsTongXunLockCommand AND VarGpsSystemLockedState,
								B6:=0,B7:=0);
		send_data300_1[2]:=PACK(B0:=NOT VarCanGpsKongZhiQiLockCommand,
								B1:=1,
								B2:=NOT VarCanGpsYanShiLockCommand ,
								B3:= NOT VarCanGpsTianXianLockCommand,
								B4:=NOT VarCanGpsKaiGaiLockCommand,
								B5:=NOT VarCanGpsTongXunLockCommand,
								B6:=0,B7:=0);
		send_data300_1[3]:=UINT_TO_USINT(CAN_NewGpsRecLockCommand);
		send_data300_1[4]:=UINT_TO_USINT(CAN_NewGpsRecUnLockCommand);
		send_data300_1[5]:=UINT_TO_USINT(CAN_TranData_NewGps1);
		send_data300_1[6]:=UINT_TO_USINT(CAN_TranData_NewGps2);
		send_data300_1[7]:=0;
		IF(VarGpsPasswordTempUnlockEnable)THEN
			CAN_TranData_NewGps1:=16#4A;
			CAN_TranData_NewGps2:=16#53;
		ELSE
			CAN_TranData_NewGps1:=16#00;
			CAN_TranData_NewGps2:=16#00;
		END_IF
	3:(*组合向GPS发送的新版协议数据,序号0x03*)
		send_data300_1[0]:=16#03;
		send_data300_1[1]:=0;
		send_data300_1[2]:=0;
		send_data300_1[3]:=0;
		send_data300_1[4]:=0;
		send_data300_1[5]:=0;
		send_data300_1[6]:=0;
		send_data300_1[7]:=0;

	4:(*组合向GPS发送的新版协议数据,序号0x04*)
		send_data300_1[0]:=16#04;
		send_data300_1[1]:=UINT_TO_USINT(CAN_NewGpsRealFakeTranData MOD 256);
		send_data300_1[2]:=UINT_TO_USINT(CAN_NewGpsRealFakeTranData/256);
		send_data300_1[3]:=UINT_TO_USINT(CANO_PowerNiuJu / 256);
		send_data300_1[4]:=UINT_TO_USINT(CANO_PowerNiuJu MOD 256);
		send_data300_1[5]:=0;
		send_data300_1[6]:=0;
		send_data300_1[7]:=0;
	5:(*组合向GPS发送的新版协议数据,序号0x05*)
		send_data300_1[0]:=16#05;
		send_data300_1[1]:=INT_TO_USINT(CANO_water_tem);
		send_data300_1[2]:=UINT_TO_USINT(CANO_Hyd_Tem);
		send_data300_1[3]:=UINT_TO_USINT(CANO_FUEL_LEVEL);
		send_data300_1[4]:=UDINT_TO_USINT((CANO_ACCMUDEPTH/100 MOD 65535) MOD 256);
		send_data300_1[5]:=UDINT_TO_USINT((CANO_ACCMUDEPTH/100 MOD 65535) /256);
		send_data300_1[6]:=UDINT_TO_USINT((CANO_ACCMUDEPTH/100 / 65535) MOD 256);
		send_data300_1[7]:=UDINT_TO_USINT((CANO_ACCMUDEPTH/100 / 65535)/256);
	6:(*组合向GPS发送的新版协议数据,序号0x06*)
		send_data300_1[0]:=16#06;
		send_data300_1[1]:=UINT_TO_USINT(CANO_Lub_Press);
		send_data300_1[2]:=PACK(B0:=CANO_TooLow_OilPress,B1:=CANO_TooHigh_WaterTem,B2:=0,B3:=CANO_TooLow_FUEL_LEVEL,B4:=0,B5:=0,B6:=0,B7:=0);
		send_data300_1[3]:=6;//V3.4版本
		send_data300_1[4]:=UDINT_TO_USINT(CANO_engine_hour_h  MOD 256);
		send_data300_1[5]:=UDINT_TO_USINT(CANO_engine_hour_h /256);
		send_data300_1[7]:=BYTE_TO_USINT(CANO_engine_hour_m);
	7:(*组合向GPS发送的新版协议数据,序号0x07*)
		send_data300_1[0]:=16#07;
		send_data300_1[1]:=UINT_TO_USINT(CANO_DonglitouPressure/10);
		send_data300_1[2]:=UINT_TO_USINT(CANO_JiayaPressure/10);
		send_data300_1[3]:=UINT_TO_USINT(CANO_ZhuJuanPressure/10);
		send_data300_1[4]:=0;
		send_data300_1[5]:=0;
		send_data300_1[6]:=0;
		send_data300_1[7]:=0;
	8:(*组合向GPS发送的新版协议数据,序号0x08*)
		send_data300_1[0]:=16#08;
		send_data300_1[1]:=UINT_TO_USINT((CANO_SPEED+1) MOD 256);
		send_data300_1[2]:=UINT_TO_USINT((CANO_SPEED+1)/256);
		send_data300_1[3]:=UINT_TO_USINT(0);
		send_data300_1[4]:=UDINT_TO_USINT((CANO_Accumu_Fuel MOD 65535) MOD 256);
		send_data300_1[5]:=UDINT_TO_USINT((CANO_Accumu_Fuel MOD 65535) /256);
		send_data300_1[6]:=UDINT_TO_USINT((CANO_Accumu_Fuel / 65535) MOD 256);
		send_data300_1[7]:=UDINT_TO_USINT((CANO_Accumu_Fuel / 65535)/256);
	9:(*组合向GPS发送的新版协议数据,序号0x09*)
		send_data300_1[0]:=16#09;
		send_data300_1[1]:=UINT_TO_USINT(CANI_JOYX_L MOD 256);
		send_data300_1[2]:=UINT_TO_USINT(CANI_JOYX_L/256);
		send_data300_1[3]:=UINT_TO_USINT(CANI_JOYY_L MOD 256);
		send_data300_1[4]:=UINT_TO_USINT(CANI_JOYY_L/256);
		send_data300_1[5]:=UINT_TO_USINT(CANI_JOYX_R MOD 256);
		send_data300_1[6]:=UINT_TO_USINT(CANI_JOYX_R/256);
		send_data300_1[7]:=UINT_TO_USINT(0/256);
	10:(*组合向GPS发送的新版协议数据,序号0x0A*)
		send_data300_1[0]:=16#0A;
		send_data300_1[1]:=UINT_TO_USINT(CANI_JOYY_R MOD 256);
		send_data300_1[2]:=UINT_TO_USINT(CANI_JOYY_R/256);
		send_data300_1[3]:=UINT_TO_USINT(CANI_JOY_Jiao_L MOD 256);
		send_data300_1[4]:=UINT_TO_USINT(CANI_JOY_Jiao_L/256);
		send_data300_1[5]:=UINT_TO_USINT(CANI_JOY_Jiao_R MOD 256);
		send_data300_1[6]:=UINT_TO_USINT(CANI_JOY_Jiao_R/256);
		send_data300_1[7]:=UINT_TO_USINT(0/256);
	11:(*组合向GPS发送的新版协议数据,序号0x0B*)
		send_data300_1[0]:=16#0B;
		send_data300_1[1]:=UINT_TO_USINT(PWM_Y1_SET MOD 256);
		send_data300_1[2]:=UINT_TO_USINT(PWM_Y1_SET/256);
		send_data300_1[3]:=UINT_TO_USINT(PWM_Y2_SET MOD 256);
		send_data300_1[4]:=UINT_TO_USINT(PWM_Y2_SET/256);
		send_data300_1[5]:=UINT_TO_USINT(PWM_Y7_SET MOD 256);
		send_data300_1[6]:=UINT_TO_USINT(PWM_Y7_SET/256);
		send_data300_1[7]:=UINT_TO_USINT(0/256);
	12:(*组合向GPS发送的新版协议数据,序号0x0C*)
		send_data300_1[0]:=16#0C;
		send_data300_1[1]:=UINT_TO_USINT(PWM_Y8_SET MOD 256);
		send_data300_1[2]:=UINT_TO_USINT(PWM_Y8_SET/256);
		send_data300_1[3]:=UINT_TO_USINT(PWM_Y9_SET MOD 256);
		send_data300_1[4]:=UINT_TO_USINT(PWM_Y9_SET/256);
		send_data300_1[5]:=UINT_TO_USINT(PWM_Y10_SET MOD 256);
		send_data300_1[6]:=UINT_TO_USINT(PWM_Y10_SET/256);
		send_data300_1[7]:=UINT_TO_USINT(0/256);
	13:(*组合向GPS发送的新版协议数据,序号0x0D*)
		send_data300_1[0]:=16#0D;
		send_data300_1[1]:=UINT_TO_USINT(PWM_Y11_SET MOD 256);
		send_data300_1[2]:=UINT_TO_USINT(PWM_Y11_SET/256);
		send_data300_1[3]:=UINT_TO_USINT(PWM_Y12_SET MOD 256);
		send_data300_1[4]:=UINT_TO_USINT(PWM_Y12_SET/256);
		send_data300_1[5]:=UINT_TO_USINT(PWM_Y13_SET MOD 256);
		send_data300_1[6]:=UINT_TO_USINT(PWM_Y13_SET/256);
		send_data300_1[7]:=UINT_TO_USINT(0/256);
	14:(*组合向GPS发送的新版协议数据,序号0x0E*)
		send_data300_1[0]:=16#0E;
		send_data300_1[1]:=UINT_TO_USINT(PWM_Y14_SET MOD 256);
		send_data300_1[2]:=UINT_TO_USINT(PWM_Y14_SET/256);
		send_data300_1[3]:=UINT_TO_USINT(PWM_Y60_SET MOD 256);
		send_data300_1[4]:=UINT_TO_USINT(PWM_Y60_SET/256);
		send_data300_1[5]:=UINT_TO_USINT(PWM_Y61_SET MOD 256);
		send_data300_1[6]:=UINT_TO_USINT(PWM_Y61_SET/256);
		send_data300_1[7]:=UINT_TO_USINT(0/256);
	15:(*组合向GPS发送的新版协议数据,序号0x0F*)
		send_data300_1[0]:=16#0F;
		send_data300_1[1]:=UINT_TO_USINT(PWM_Y23_SET MOD 256);
		send_data300_1[2]:=UINT_TO_USINT(PWM_Y23_SET/256);
		send_data300_1[3]:=UINT_TO_USINT(PWM_Y24_SET MOD 256);
		send_data300_1[4]:=UINT_TO_USINT(PWM_Y24_SET/256);
		send_data300_1[5]:=UINT_TO_USINT(PWM_Y21_SET MOD 256);
		send_data300_1[6]:=UINT_TO_USINT(PWM_Y21_SET/256);
		send_data300_1[7]:=UINT_TO_USINT(0/256);
	16:(*组合向GPS发送的新版协议数据,序号0x10*)
		send_data300_1[0]:=16#10;
		send_data300_1[1]:=UINT_TO_USINT(CANO_MainWinch_Speed MOD 256 );
		send_data300_1[2]:=UINT_TO_USINT(CANO_MainWinch_Speed/256);
		send_data300_1[3]:=UINT_TO_USINT(CANO_DEPTH MOD 256 );
		send_data300_1[4]:=UINT_TO_USINT(CANO_DEPTH/256);
		send_data300_1[5]:=BOOL_TO_USINT(CANI_Button_RecordClear);
		send_data300_1[6]:=UINT_TO_USINT(FuelMomentary MOD 256 );
		send_data300_1[7]:=UINT_TO_USINT(FuelMomentary/256);
	17:(*组合向GPS发送的新版协议数据,序号0x11*)
		send_data300_1[0]:=16#11;
		send_data300_1[1]:=UINT_TO_USINT(CANO_ANGLE_X MOD 256 );
		send_data300_1[2]:=UINT_TO_USINT(CANO_ANGLE_X/256);
		send_data300_1[3]:=UINT_TO_USINT(CANO_ANGLE_Y MOD 256 );
		send_data300_1[4]:=UINT_TO_USINT(CANO_ANGLE_Y/256);
		send_data300_1[5]:=PACK(B0:=DI_LHandle_SB2,B1:=VarMastAutoEnable,B2:=DOH_Y55,B3:= 0,
								B4:=0,B5:=0,B6:=0,B7:=0);
		send_data300_1[6]:=UINT_TO_USINT(VarMastLimitState);
		send_data300_1[7]:=UINT_TO_USINT(CANO_PilotPressure);
	18:(*组合向GPS发送的新版协议数据,序号0x12*)
		send_data300_1[0]:=16#12;
		send_data300_1[1]:=UINT_TO_USINT(0 MOD 256 );
		send_data300_1[2]:=UINT_TO_USINT(0/256);
		send_data300_1[3]:=UINT_TO_USINT(PileNumble / 256 );
		send_data300_1[4]:=UINT_TO_USINT(PileNumble MOD 256);
		send_data300_1[5]:=UINT_TO_USINT(PileDiameter / 256 );
		send_data300_1[6]:=UINT_TO_USINT(PileDiameter MOD 256);
		send_data300_1[7]:=UINT_TO_USINT(CANO_PowerSpeed);
	19:(*组合向GPS发送的新版协议数据,序号0x13*)
		send_data300_1[0]:=16#13;
		send_data300_1[1]:=UINT_TO_USINT(X_Offset / 256 );
		send_data300_1[2]:=UINT_TO_USINT(X_Offset MOD 256);
		send_data300_1[3]:=UINT_TO_USINT(Y_Offset / 256 );
		send_data300_1[4]:=UINT_TO_USINT(Y_Offset MOD 256);
		send_data300_1[5]:=UINT_TO_USINT(0 / 256 );
		send_data300_1[6]:=UINT_TO_USINT(0 MOD 256);
		send_data300_1[7]:=UINT_TO_USINT(0);
	20:(*组合向GPS发送的新版协议数据,序号0x14*)
		send_data300_1[0]:=16#14;
		send_data300_1[1]:=UINT_TO_USINT(PWM_Y22_SET MOD 256);
		send_data300_1[2]:=UINT_TO_USINT(PWM_Y22_SET/256);
		send_data300_1[3]:=UINT_TO_USINT(PWM_Y5_SET MOD 256);
		send_data300_1[4]:=UINT_TO_USINT(PWM_Y5_SET/256);
		send_data300_1[5]:=UINT_TO_USINT(PWM_Y6_SET MOD 256);
		send_data300_1[6]:=UINT_TO_USINT(PWM_Y6_SET/256);
		send_data300_1[7]:=UINT_TO_USINT(0/256);
	21:(*组合向GPS发送的新版协议数据,序号0x15*)
		send_data300_1[0]:=16#15;
		send_data300_1[1]:=UINT_TO_USINT(PWM_Y34_SET MOD 256);
		send_data300_1[2]:=UINT_TO_USINT(PWM_Y34_SET/256);
		send_data300_1[3]:=UINT_TO_USINT(PWM_Y33_SET MOD 256);
		send_data300_1[4]:=UINT_TO_USINT(PWM_Y33_SET/256);
		send_data300_1[5]:=UINT_TO_USINT(PWM_Y39_SET MOD 256);
		send_data300_1[6]:=UINT_TO_USINT(PWM_Y39_SET/256);
		send_data300_1[7]:=PACK(B0:=DI_LHandle_SB1,B1:=DI_LHandle_SB2,B2:=DI_LHandle_SB3,B3:= DI_LHandle_SB4,
								B4:=DI_RHandle_SB5,B5:=DI_RHandle_SB6,B6:=DI_RHandle_SB8A,B7:=DI_RHandle_SB8B);
	22:(*组合向GPS发送的新版协议数据,序号0x16*)
		send_data300_1[0]:=16#16;
		send_data300_1[1]:=UINT_TO_USINT(PWM_Y40_SET MOD 256);
		send_data300_1[2]:=UINT_TO_USINT(PWM_Y40_SET/256);
		send_data300_1[3]:=UINT_TO_USINT(DI_LHandle_SB4_UINT MOD 256);
		send_data300_1[4]:=UINT_TO_USINT(DI_LHandle_SB4_UINT/256);
		send_data300_1[5]:=UINT_TO_USINT(DI_RHandle_SB7_UINT MOD 256);
		send_data300_1[6]:=UINT_TO_USINT(DI_RHandle_SB7_UINT/256);
		send_data300_1[7]:=0;
END_CASE

send_data300[0]:= NOT send_data300_1[0];
send_data300[1]:= NOT send_data300_1[1];
send_data300[2]:= NOT send_data300_1[2];
send_data300[3]:= NOT send_data300_1[3];
send_data300[4]:= NOT send_data300_1[4];
send_data300[5]:= NOT send_data300_1[5];
send_data300[6]:= NOT send_data300_1[6];
send_data300[7]:= NOT send_data300_1[7];
CAN2_SEND_300(xEnable:= TRUE, eChannel:= 1, udiID:= 16#300, xExtended:=FALSE, usiDLC:=8 , aData:=send_data300 );


(*控制器接受GPS数据*)
CAN2_RECE_GPS200(xEnable:=TRUE , eChannel:= 1, xExtended:= FALSE, aData=> receive_data200, udiID:= 16#200);
receive_data200[0]:=NOT receive_data200[0];
receive_data200[1]:=NOT receive_data200[1];
receive_data200[2]:=NOT receive_data200[2];
receive_data200[3]:=NOT receive_data200[3];
receive_data200[4]:=NOT receive_data200[4];
receive_data200[5]:=NOT receive_data200[5];
receive_data200[6]:=NOT receive_data200[6];
receive_data200[7]:=NOT receive_data200[7];
CASE  receive_data200[0] OF
	0:
		VarCanNewGpsVersion:=receive_data200[2]+256*receive_data200[3];
		VarCanNewGpsManufacturers:=receive_data200[4];
	1:;
	2:
		VarCanNewGpsRecLockCommand:=receive_data200[1];
		VarCanNewGpsRecUnlockCommand:=receive_data200[2];
		IF(receive_data200[3]=1)THEN//网络临时解锁指令
			VarGpsPasswordTempUnlockCount:=VarGpsPasswordTempUnlockCount+1;
			IF(VarGpsPasswordTempUnlockCount>=5)THEN
				VarGpsPasswordTempUnlockCount:=0;
				IF(NOT VarGpsPasswordTempUnlockEnable)THEN
					VarGpsPasswordTempUnlockEnable:=TRUE;
				END_IF
			END_IF
		ELSIF(receive_data200[3]=0)THEN
			VarGpsPasswordTempUnlockCount:=0;
		END_IF;
		IF(BYTE_TO_BOOL(receive_data200[1] AND 2#00000001) AND NOT BYTE_TO_BOOL(receive_data200[2] AND 2#00000001))THEN
			VarCanGpsKongZhiQiLockCommand:=TRUE;
		ELSIF(BYTE_TO_BOOL (receive_data200[2] AND 2#00000001)AND NOT BYTE_TO_BOOL (receive_data200[1] AND 2#00000001))THEN
			VarCanGpsKongZhiQiLockCommand:=FALSE;
		END_IF
	(*	IF(BYTE_TO_BOOL (receive_data200[1] AND 2#00000100) AND NOT BYTE_TO_BOOL(receive_data200[2] AND 2#00000100))THEN
			VarCanGpsYanShiLockCommand:=TRUE;
		ELSIF(BYTE_TO_BOOL (receive_data200[2] AND 2#00000100)AND NOT BYTE_TO_BOOL (receive_data200[1] AND 2#00000100))THEN
			VarCanGpsYanShiLockCommand:=FALSE;
		END_IF*)
		IF(BYTE_TO_BOOL (receive_data200[1] AND 2#00001000) AND NOT BYTE_TO_BOOL (receive_data200[2] AND 2#00001000))THEN
			VarCanGpsTianXianLockCommand:=TRUE;
		ELSIF(BYTE_TO_BOOL(receive_data200[2] AND 2#00001000)AND NOT BYTE_TO_BOOL (receive_data200[1] AND 2#00001000))THEN
			VarCanGpsTianXianLockCommand:=FALSE;
		END_IF
		IF(BYTE_TO_BOOL (receive_data200[1] AND 2#00010000) AND NOT BYTE_TO_BOOL (receive_data200[2] AND 2#00010000))THEN
			VarCanGpsKaiGaiLockCommand:=TRUE;
		ELSIF(BYTE_TO_BOOL (receive_data200[2] AND 2#00010000)AND NOT BYTE_TO_BOOL (receive_data200[1] AND 2#00010000))THEN
			VarCanGpsKaiGaiLockCommand:=FALSE;
		END_IF
		
		IF (BYTE_TO_BOOL (receive_data200[1] AND 2#00100000)) THEN
			VarCanNewGpsNoSignalLock_Warning:=TRUE;
		ELSE
			VarCanNewGpsNoSignalLock_Warning:=FALSE;
		END_IF
	3:;
	4:	
		VarCanNewGpsRealFakeRecData:=receive_data200[1]+256*receive_data200[2];
	5:;
	6:;
	7:;
	8: 
		GPS_Time_bool:=USINT_TO_BOOL(receive_data200[1]);
		GPS_Time_Year:=receive_data200[2];
		GPS_Time_Month:=receive_data200[2];
		GPS_Time_Day:=receive_data200[2];
		GPS_Time_Hour:=receive_data200[2];
		GPS_Time_Minute:=receive_data200[2];
		GPS_Time_Second:=receive_data200[2];
	9:
		GPS_Signal_Intensity:=receive_data200[1];
END_CASE


send_data18FF0001[0]:=UINT_TO_USINT(Time_Minute_Left MOD 256);
send_data18FF0001[1]:=UINT_TO_USINT(Time_Minute_Left / 256);
send_data18FF0001[2]:=PACK(B0:=VarCanNewGpsNoSignalLock_Warning,
						   B1:=(VarGpsSystemLockedState_bool OR (VarCanGpsTongXunLockCommand AND VarGpsGlobalEnable)),
						   B2:=VarGpsSystemLockedState,B3:=0,
						   B4:=0,B5:=0,B6:=0,B7:=0);
send_data18FF0001[3]:=GPS_Signal_Intensity;
send_data18FF0001[4]:=0;
send_data18FF0001[5]:=0;
send_data18FF0001[6]:=0;
send_data18FF0001[7]:=0;
CAN2_SEND_18FF00001(xEnable:= TRUE, eChannel:= 0, udiID:= 16#18FF0001, xExtended:=TRUE, usiDLC:=8 , aData:=send_data18FF0001 );


(***GPS 锁车***)
(***拆除GPS****)
IF(CAN2_RECE_GPS200.uiAvailable=0)THEN
	GPS_CAN_ERROR_1:=TRUE;
ELSE
	GPS_CAN_ERROR_1:=FALSE;
END_IF
TIME_2s(IN:=NOT TIME_2s.Q,PT:=T#2S);
IF(TIME_2s.Q)THEN
	IF(VarCanGpsTongXunLockErrorTimer2S<1000) AND GPS_CAN_ERROR_1 THEN	
		VarCanGpsTongXunLockErrorTimer2S:=VarCanGpsTongXunLockErrorTimer2S+1;
		IF(VarCanGpsTongXunLockErrorTimer2S>150)THEN     //5分钟
			VarCanGpsTongXunLockCommand:=TRUE;
			VarCanGpsTongXunLockErrorTimer2S:=0;
		END_IF
	END_IF
END_IF
IF NOT GPS_CAN_ERROR_1 THEN
		VarCanGpsTongXunLockCommand:=FALSE;
		VarCanGpsTongXunLockErrorTimer2S:=0;
END_IF
(***假GPS****)
(**随机生成真假GPS识别数据,此数据用于发送给GPS**)
TIME_600S(IN:=NOT TIME_600S.Q,PT:=T#600S);
IF	TIME_600S.Q  THEN
	CAN_NewGpsRealFakeTranData:=CANO_VOL_VALUE+INT_TO_UINT(CANO_water_tem);
END_IF
TIME_1S(IN:=NOT TIME_1S.Q,PT:=T#1S);
IF	TIME_1S.Q  THEN
	tU8_H:=UINT_TO_USINT(CAN_NewGpsRealFakeTranData MOD 256);
	tU8_L:=UINT_TO_USINT(CAN_NewGpsRealFakeTranData/256);
	tU16:=tU8_H*256+tU8_L;
	tU16:=tU16+CANO_engine_hour_m;
	IF	CANO_engine_hour_m>=30 THEN
		tU16:=NOT tU16 ;
		VarCanNewGpsRealFakeTargetData:=tU16;
	ELSE
		tU8_H:=UINT_TO_USINT(tU16 MOD 256);
		tU8_L:=UINT_TO_USINT(tU16 / 256);
		VarCanNewGpsRealFakeTargetData:=tU8_H*256+tU8_L;
	END_IF
	IF(VarCanNewGpsRealFakeTargetData =VarCanNewGpsRealFakeRecData)THEN
		VarCanNewGpsRealFakeResult:=TRUE;
	ELSE
		VarCanNewGpsRealFakeResult:=FALSE;
	END_IF
END_IF
TIME_1S_1(IN:=NOT TIME_1S_1.Q,PT:=T#1S);
IF(TIME_1S_1.Q)THEN
	IF(VarCanGpsFakeErrorTimer1S<1000) AND NOT VarCanNewGpsRealFakeResult THEN
		VarCanGpsFakeErrorTimer1S:=VarCanGpsFakeErrorTimer1S+1;
		IF(VarCanGpsFakeErrorTimer1S>60)THEN  //1分钟
				VarCanGpsFakeLockCommand:=TRUE;
				VarCanGpsFakeErrorTimer1S:=0;
		END_IF
	END_IF
END_IF
IF(VarCanNewGpsRealFakeResult)THEN
		VarCanGpsFakeLockCommand:=FALSE;
		VarCanGpsFakeErrorTimer1S:=0;
	END_IF
(***所有条件的锁GPS****)
IF(VarGpsGlobalEnable AND  NOT VarGpsTempUnlockDoing AND NOT VarGpsPasswordTempUnlockEnable)THEN    //锁车全局使能并且没有临时解锁
	IF(VarCanGpsKongZhiQiLockCommand  OR VarCanGpsTianXianLockCommand OR
		VarCanGpsKaiGaiLockCommand )THEN
			VarGpsSystemLockedState:=TRUE;
	ELSIF(VarCanGpsTongXunLockCommand OR VarCanGpsFakeLockCommand) THEN
			VarGpsSystemLockedState:=TRUE;
	ELSE
		VarGpsSystemLockedState:=FALSE;
		VarGpsSystemLockedState_bool:=FALSE;
	END_IF
ELSE
	VarGpsSystemLockedState:=FALSE;
	VarGpsSystemLockedState_bool:=FALSE;
END_IF

	//延时2小时锁车
	IF((NOT VarGpsSystemLockedState) AND VarGpsSystemLockedState_bool) THEN//已下锁车指令 无锁车时运行
		IF(VarGpsSystemLockedState_bool AND Time_bool_once) THEN
			GPS_Time_Year_Last := GPS_Time_Year;
			GPS_Time_Month_Last := GPS_Time_Month;
			GPS_Time_Day_Last  :=  GPS_Time_Day;
			GPS_Time_Hour_Last := GPS_Time_Hour;
			GPS_Time_Minute_Last := GPS_Time_Minute;
			GPS_Time_Second_Last := GPS_Time_Second;
			Time_bool_once := FALSE;
		END_IF
				
		IF(GPS_Time_Year>=GPS_Time_Year_Last)THEN
			Time_Sub_Year := GPS_Time_Year - GPS_Time_Year_Last;		
		END_IF
		IF(GPS_Time_Month>=GPS_Time_Month_Last)THEN
			Time_Sub_Month := GPS_Time_Month - GPS_Time_Month_Last;		
		END_IF
		IF(GPS_Time_Day>=GPS_Time_Day_Last) THEN
			Time_Sub_Day := GPS_Time_Day - GPS_Time_Day_Last;		
		END_IF
		
		IF(Time_Sub_Day=1 OR Time_Sub_Year=1 OR Time_Sub_Month=1) THEN
			Time_Sub_Hour := 24 - GPS_Time_Hour_Last + GPS_Time_Hour;
		ELSIF(Time_Sub_Day>1)THEN
			Time_Sub_Hour := 24;
		ELSE
			Time_Sub_Hour := GPS_Time_Hour - GPS_Time_Hour_Last;
		END_IF
		
		IF(GPS_Time_bool) THEN
			Time_Minute_Left := 360 - Time_Sub_Hour * 60 - GPS_Time_Minute + GPS_Time_Minute_Last;
		END_IF
			
		IF(Time_Minute_Left>360) THEN
			Time_Minute_Left := 0;
		END_IF
		
		IF(Time_Minute_Left = 0) THEN
			VarGpsSystemLockedState := TRUE;
		END_IF
	END_IF
		
	IF((NOT VarGpsSystemLockedState_bool) AND (NOT Time_bool_once)) THEN
		Time_bool_once := TRUE;
	END_IF

	
(***GPS 解锁***)
(***网络临时解锁计时***)
TIME_60S(IN:=NOT TIME_60S.Q,PT:=T#60S);
IF(TIME_60S.Q)THEN
	IF(VarGpsPasswordTempUnlockTimer60S<2000) AND VarGpsPasswordTempUnlockEnable  THEN
		VarGpsPasswordTempUnlockTimer60S:=VarGpsPasswordTempUnlockTimer60S+1;
		IF(VarGpsPasswordTempUnlockTimer60S>1440) THEN
			VarGpsPasswordTempUnlockEnable:=FALSE;
			VarGpsPasswordTempUnlockTimer60S:=0;
		END_IF
	END_IF
	IF(VarGpsPasswordTemporaryCode=9996) AND VarGpsPasswordTempUnlockEnable THEN
		VarGpsPasswordTempUnlockEnable:=FALSE;
		VarGpsPasswordTempUnlockTimer60S:=0;
	END_IF
END_IF
(***本地临时解锁*****)
IF(VarGpsGlobalEnable)THEN
	IF(VarGpsTempUnlockPassword=9996 AND BYTE_TO_BOOL(VarGpsTempUnlockSelect AND 2#11111111))THEN
		VarGpsTempUnlockSelect:=0;
		VarGpsPasswordTempUnlockTimer60S:=0;
	ELSIF(VarGpsTempUnlockPassword=8402 AND BYTE_TO_BOOL(VarGpsTempUnlockEnable AND 2#00000001))THEN
		VarGpsTempUnlockSelect:=VarGpsTempUnlockSelect OR 2#00000001;
        VarGpsTempUnlockEnable:= VarGpsTempUnlockEnable AND  2#11111110;
	ELSIF(VarGpsTempUnlockPassword=6308 AND BYTE_TO_BOOL(VarGpsTempUnlockEnable AND 2#00000010))THEN
		VarGpsTempUnlockSelect:=VarGpsTempUnlockSelect OR 2#00000010;
        VarGpsTempUnlockEnable:= VarGpsTempUnlockEnable AND  2#11111101;
	ELSIF(VarGpsTempUnlockPassword=8815 AND BYTE_TO_BOOL(VarGpsTempUnlockEnable AND 2#00000100))THEN
		VarGpsTempUnlockSelect:=VarGpsTempUnlockSelect OR 2#00000100;
        VarGpsTempUnlockEnable:= VarGpsTempUnlockEnable AND  2#11111011;
	ELSIF(VarGpsTempUnlockPassword=1678 AND BYTE_TO_BOOL(VarGpsTempUnlockEnable AND 2#00001000))THEN
		VarGpsTempUnlockSelect:=VarGpsTempUnlockSelect OR 2#00001000;
        VarGpsTempUnlockEnable:= VarGpsTempUnlockEnable AND  2#11110111;
	ELSIF(VarGpsTempUnlockPassword=9854 AND BYTE_TO_BOOL(VarGpsTempUnlockEnable AND 2#00010000))THEN
		VarGpsTempUnlockSelect:=VarGpsTempUnlockSelect OR 2#00010000;
        VarGpsTempUnlockEnable:= VarGpsTempUnlockEnable AND  2#11101111;
	ELSIF(VarGpsTempUnlockPassword=11345 AND BYTE_TO_BOOL(VarGpsTempUnlockEnable AND 2#00100000))THEN
		VarGpsTempUnlockSelect:=VarGpsTempUnlockSelect OR 2#00100000;
        VarGpsTempUnlockEnable:= VarGpsTempUnlockEnable AND  2#11011111;
	ELSIF(VarGpsTempUnlockPassword=15342 AND BYTE_TO_BOOL(VarGpsTempUnlockEnable AND 2#01000000))THEN
		VarGpsTempUnlockSelect:=VarGpsTempUnlockSelect OR 2#01000000;
        VarGpsTempUnlockEnable:= VarGpsTempUnlockEnable AND  2#10111111;
	ELSIF(VarGpsTempUnlockPassword=26742 AND BYTE_TO_BOOL(VarGpsTempUnlockEnable AND 2#10000000))THEN
		VarGpsTempUnlockSelect:=VarGpsTempUnlockSelect OR 2#10000000;
        VarGpsTempUnlockEnable:= VarGpsTempUnlockEnable AND  2#01111111;
	END_IF
END_IF
IF(BYTE_TO_BOOL(VarGpsTempUnlockSelect AND 2#11111111) AND VarGpsGlobalEnable)THEN
	IF(VarGpsPasswordTempUnlockTimer60S<=1440)THEN
		VarGpsTempUnlockDoing:=TRUE;
	ELSE
		VarGpsTempUnlockDoing:=FALSE;
		VarGpsTempUnlockSelect:=0;
		VarGpsPasswordTempUnlockTimer60S:=0;
	END_IF
ELSE
	VarGpsTempUnlockDoing:=FALSE;
END_IF
TIME_60s_2(IN:=NOT TIME_60s_2.Q,PT:=T#60S);
IF(TIME_60s_2.Q)THEN
	IF(VarGpsPasswordTempUnlockTimer60S<2000) AND VarGpsTempUnlockDoing    THEN
		VarGpsPasswordTempUnlockTimer60S:=VarGpsPasswordTempUnlockTimer60S+1;
	END_IF
END_IF
(***永久解锁*****)
GPSYONGJIU(
	Engine_Hour:= UDINT_TO_DINT(CANO_engine_hour_h), 
	Engine_Minute:=CANO_engine_hour_m , 
	Accum_Depth:= UDINT_TO_DINT(CANO_ACCMUDEPTH)/100, 
	Hyhoil_Tem:= CANO_Hyd_Tem, 
	Water_Tem:=CANO_water_tem , 
	PassWard=> VarGpsYongJiuUnlockPassword);

IF (PAR_GPS_ForeverUnlockPassword=VarGpsYongJiuUnlockPassword)THEN
	IF(VarGpsGlobalEnable)THEN
		VarGpsGlobalEnable:=FALSE;
	END_IF
ELSIF(PAR_GPS_ForeverUnlockPassword=9996)THEN
	IF(NOT VarGpsGlobalEnable)THEN
		VarGpsGlobalEnable:=TRUE;
	END_IF
END_IF

END_PROGRAM

// Project Information/GetTextProperty
// This function has been automatically generated from the project information.
{attribute 'signature_flag' := '1073741824'}
{attribute 'register_in_runtime'}
FUNCTION GetTextProperty : WSTRING
VAR_INPUT
	stKey: WSTRING;
END_VAR

IF stKey = "Company" THEN
	GetTextProperty := "ifm electronic";
ELSIF stKey = "Description" THEN
	GetTextProperty := "CR721S 2.25MByte Standard and Safety";
ELSIF stKey = "Project" THEN
	GetTextProperty := "SWDM240HES_S00107_20240126_Y33";
ELSIF stKey = "Title" THEN
	GetTextProperty := "ifmCR721S_TemplateProject";
ELSE
	GetTextProperty := "";
END_IF

END_FUNCTION

// Project Information/GetBooleanProperty
// This function has been automatically generated from the project information.
{attribute 'signature_flag' := '1073741824'}
{attribute 'register_in_runtime'}
FUNCTION GetBooleanProperty : BOOL
VAR_INPUT
	stKey: WSTRING;
END_VAR

IF stKey = "Released" THEN
	GetBooleanProperty := FALSE;
ELSE
	GetBooleanProperty := FALSE;
END_IF

END_FUNCTION

// Project Information/GetVersionProperty
// This function has been automatically generated from the project information.
{attribute 'signature_flag' := '1073741824'}
{attribute 'register_in_runtime'}
FUNCTION GetVersionProperty : VERSION
VAR_INPUT
	stKey: WSTRING;
END_VAR

IF stKey = "Version" THEN
	GetVersionProperty.uiMajor := 3;
	GetVersionProperty.uiMinor := 1;
	GetVersionProperty.uiServicePack := 4;
	GetVersionProperty.uiPatch := 1;
ELSE
	GetVersionProperty.uiMajor := 0;
	GetVersionProperty.uiMinor := 0;
	GetVersionProperty.uiServicePack := 0;
	GetVersionProperty.uiPatch := 0;
END_IF

END_FUNCTION

// Project Information/GetNumberProperty
// This function has been automatically generated from the project information.
{attribute 'signature_flag' := '1073741824'}
{attribute 'register_in_runtime'}
FUNCTION GetNumberProperty : DINT
VAR_INPUT
	stKey: WSTRING;
END_VAR

GetNumberProperty := 0;

END_FUNCTION

// StandardPLC/Application/SaveEngine/SaveEngineMode_19
PROGRAM SaveEngineMode_19
VAR

END_VAR

(*******************节能控制阀主阀主泵输出执行**************************)

END_PROGRAM
